TYPE Sfts_Control_DUT :
STRUCT
	Mode:  UINT;
	Error:  BOOL;
	Enabled:  Bool;
	Running:  Bool;
	LP_State:  USInt;
	Motor_Extend:  Bool;
	Motor_Retract:  Bool;
	SM_State:  UInt;
	Instruction:  Sfts_Instruction_DUT;
	Inputs:  Sfts_Inputs_DUT;
END_STRUCT
END_TYPE

(* stored: Version 1.1.0.1
   DUT Sfts_Control_DUT: Id {521028b3-7fc6-4f9d-97cf-0c6b505fc9b2} *)
